{attribute 'linkalways'} 
{attribute 'no_explicit_call' := 'This FB is a CLASS and must be accessed using methods or properties'}
{attribute 'enable_dynamic_creation'}
FUNCTION_BLOCK FINAL SEL_LINT EXTENDS Node
VAR
	g : _BOOL(FALSE);
	in1 : _LINT(0);
	in2 : _LINT(0);
	out : _LINT(0);
END_VAR

METHOD PUBLIC Clone : I_Node
VAR
	pNode : POINTER TO SEL_LINT;
END_VAR
pNode := __NEW(SEL_LINT);
Clone := pNode^;
END_METHOD

METHOD FB_init : BOOL
VAR_INPUT
	bInitRetains : BOOL; // if TRUE, the retain variables are initialized (warm start / cold start)
	bInCopyCode : BOOL;  // if TRUE, the instance afterwards gets moved into the copy code (online change)
END_VAR
AddInput('g',THIS^.g);
AddInput('in1',THIS^.in1);
AddInput('in2',THIS^.in2);
AddOutput('out', THIS^.out);
END_METHOD

METHOD PROTECTED OnExecute
VAR
END_VAR
IF g.value THEN
	out.value := in2.value;
ELSE
	out.value := in1.value;
END_IF
END_METHOD

END_FUNCTION_BLOCK

(* stored: Version 1.1.0.1, ProductVersion 3.1.4024.15
   POU SEL_LINT: Id {612ba361-1ec6-4323-9229-472bc2b58ed8}, SpecialFunc None
   Folder Constructor: Id {e0e2ff8e-19b5-4fad-bf1b-da00d74393fe}
   Method Clone: Id {b1e8c93b-f9ac-450d-aede-cb683249fa2a}
   Method FB_init: Id {4069ce3e-7e59-495e-80bc-4a26745e55c2}
   Method OnExecute: Id {8a19b5c5-905f-4b6b-a766-d2ef6b84b2c4} *)
